INTERFACE I_IoDevice EXTENDS I_Base

{attribute 'monitoring' := 'call'}
PROPERTY IoDataValid : BOOL
GET
END_GET
END_PROPERTY

END_INTERFACE

(* stored: Version 1.1.0.1, ProductVersion 3.1.4026.18
   Itf I_IoDevice: Id {55569bad-0315-4b40-b972-0142acab1cd9}
   Property IoDataValid: Id {8281629a-37fa-44ae-b2b6-da055b34c7a5}
   Get Get: Id {b0ff3aed-ebb6-4c28-a97f-44733f96ef75} *)
